// TIA Portal project "LABSDAMC" (V20)

(* hardware
DEVICE "S7-1500/ET200MP station_1"  S7-1500 station
   slot 0: "Rail_0"  Rack  6ES7 590-1***0-0AA0
   slot 1: "PLC_1"  CPU 1516-3 PN/DP  6ES7 516-3AN01-0AB0  V2.9
      slot 3: "CPU display_1"  6ES7591-1BA00-0AA0
      slot 32768: "PROFINET interface_1"  X1
         slot 32769: "Port_1"  X1 P1
         slot 32770: "Port_2"  X1 P2
      slot 33024: "PROFINET interface_2"  X2
         slot 33025: "Port_1"  X2 P1
      slot 33280: "DP interface_1"  X3
      slot 34817: "Virtual CP interface port_1"  Virtual CP interface port  Virtual CP interface port
   slot 2: "DI 32x24VDC HF_1"  DI 32x24VDC HF  6ES7 521-1BL00-0AB0  V2.2
   slot 3: "DQ 32x24VDC/0.5A HF_1"  DQ 32x24VDC/0.5A HF  6ES7 522-1BL01-0AB0  V1.1
   slot 4: "AI 8xU/I/RTD/TC ST_1"  AI 8xU/I/RTD/TC ST  6ES7 531-7KF00-0AB0  V2.2
   slot 5: "AQ 4xU/I ST_1"  AQ 4xU/I ST  6ES7 532-5HD00-0AB0  V2.2
DEVICE "HMI"  TP900 Comfort
   slot 0: "HMI"  TP900 Comfort  6AV2 124-0JC01-0AX0  17.0.0.0
   slot 1: "HMI_RT_1"  TP900 Comfort  6AV2 124-0JC01-0AX0  17.0.0.0
   slot 5: "HMI.IE_CP_1"  PROFINET Interface  17.0.0.0
      slot 1: "PROFINET Interface_1"  PROFINET Interface
         slot 1: "Port_1"  Port
         slot 2: "Port_2"  Port
   slot 7: "HMI.MPI/DP_CP_1"  MPI/DP Interface  17.0.0.0
*)

// ===== PLC "PLC_1"  CPU 1516-3 PN/DP =====

VAR_GLOBAL   // PLC tag table "Default tag table"
   "Conveyor_Start_Backward" AT %Q0.1 : Bool;
END_VAR

VAR_GLOBAL   // PLC tag table "Tags GRAPH Sequence"
   "GRAPH_Group_Fault" AT %M10.0 : Bool;
   "GRAPH_Count_Bottle" AT %MW12 : Int;
   "Valve_water" AT %Q1.1 : Bool;
   "Valve_AJC" AT %Q1.2 : Bool;
   "Valve_OJC" AT %Q1.3 : Bool;
   "GRAPH_Mixer_ON" AT %Q1.0 : Bool;
   "GRAPH_Start_Labeling" AT %Q2.0 : Bool;
   "GRAPH_Filling_Complete" AT %M20.0 : Bool;
   "Start_GRAPH_Sequence" AT %M100.0 : Bool;
END_VAR

VAR_GLOBAL   // PLC tag table "Tag-uri de umplere"
   "Valve_Fill_Bottle" AT %Q1.4 : Bool;
END_VAR

VAR_GLOBAL   // PLC tag table "Tag-uri transport"
   "Conveyor_Direction" AT %M0.1 : Bool;
   "Conveyor_Start_Conveyor" AT %M0.0 : Bool;
   "Conveyor_Drive_OK" AT %M0.2 : Bool;
   "Conveyor_Start_Forward" AT %Q0.0 : Bool;
END_VAR

VAR_GLOBAL   // PLC tag table "Tag-uri expirare"
   "Best_before_date" AT %MW2 : Int;
END_VAR

DATA_BLOCK "Global_DB"   // DB1
{ S7_Optimized_Access := 'TRUE' }
VERSION : 0.1
   VAR
      BBD_Duration : Int;
      Rețetă_element_concentrat_suc_de_mere : Time;
      Rețetă_element_concentrat_suc_orange : Time;
      Rețetă_element_apă : Time;
   END_VAR
BEGIN
END_DATA_BLOCK

DATA_BLOCK "SetareData"   // DB2
{ S7_Optimized_Access := 'TRUE' }
VERSION : 0.1
   VAR
      data : DTL;
      ok : Int;
      data_temp : DTL;
   END_VAR
BEGIN
END_DATA_BLOCK

DATA_BLOCK "SCL_Best_before_date_DB"   // DB4
{ S7_Optimized_Access := 'TRUE' }
VERSION : 0.1
// stored: InstanceOfName SCL_Best_before_date
"SCL_Best_before_date"
BEGIN
END_DATA_BLOCK

DATA_BLOCK "GRAPH_Sequence_DB_1"   // DB5
{ S7_Optimized_Access := 'TRUE' }
VERSION : 0.1
// stored: InstanceOfName GRAPH_Sequence
"GRAPH_Sequence"
BEGIN
END_DATA_BLOCK

FUNCTION_BLOCK "GRAPH_Sequence"   // FB1, GRAPH_PLUS
{ S7_Optimized_Access := 'TRUE' }
VERSION : 0.1
   VAR_INPUT
      OFF_SQ : Bool := false;   // Turn sequence off
      INIT_SQ : Bool := false;   // Set sequence to initial state
      ACK_EF : Bool := false;   // Acknowledge all errors and faults
      S_PREV : Bool := false;   // Output previous step in parameter S_NO
      S_NEXT : Bool := false;   // Indicate next step in parameter S_NO
      SW_AUTO : Bool := false;   // Automatic mode
      SW_TAP : Bool := false;   // Semiautomatic/switch with transition
      SW_TOP : Bool := false;   // Semiautomatic/ignore transition
      SW_MAN : Bool := false;   // Manual mode
      S_SEL : Int := 0;   // Select step to be output to S_NO
      S_ON : Bool := false;   // Activate step indicated in S_NO
      S_OFF : Bool := false;   // Disable step indicated in S_NO
      T_PUSH : Bool := false;   // Enable transition to switch in semi automatic mode
   END_VAR
   VAR_OUTPUT
      S_NO : Int := 0;   // Step number
      S_MORE : Bool := false;   // More steps are available and can be shown in S_NO
      S_ACTIVE : Bool := false;   // Step indicated in S_NO is active
      ERR_FLT : Bool := false;   // Interlock or supervision group error
      AUTO_ON : Bool := false;   // Automatic mode is active
      TAP_ON : Bool := false;   // Semiautomatic mode/step with transition enabled
      TOP_ON : Bool := false;   // Semiautomatic mode/ignore transition enabled
      MAN_ON : Bool := false;   // Manual mode is active
   END_VAR
   VAR
      HMI_INFO : Array[0..8] of UInt;
      IF_PAR : G7_IfParPlus_V6;
      RT_DATA : G7_RTDataPlus_V6;   // Internal data area
      Trans1 : G7_TransitionPlus_V6;   // Transition structure
      Trans2 : G7_TransitionPlus_V6;   // Transition structure
      Trans3 : G7_TransitionPlus_V6;   // Transition structure
      Trans4 : G7_TransitionPlus_V6;   // Transition structure
      Trans5 : G7_TransitionPlus_V6;   // Transition structure
      Trans6 : G7_TransitionPlus_V6;   // Transition structure
      Trans7 : G7_TransitionPlus_V6;   // Transition structure
      Trans8 : G7_TransitionPlus_V6;   // Transition structure
      Trans9 : G7_TransitionPlus_V6;   // Transition structure
      Home : G7_StepPlus_V6;   // Step structure
      "Umpleți ingredientele rețetei" : G7_StepPlus_V6;   // Step structure
      Mixer : G7_StepPlus_V6;   // Step structure
      "Transport de umplere" : G7_StepPlus_V6;   // Step structure
      Umplere : G7_StepPlus_V6;   // Step structure
      "Etichetarea transportului" : G7_StepPlus_V6;   // Step structure
      Etichetarea : G7_StepPlus_V6;   // Step structure
      "Umplere completă" : G7_StepPlus_V6;   // Step structure
      SINI : Array[0..1] of USInt;
      LSTT : Array[0..8] of USInt;
      ATAJ : Array[0..8] of USInt;
      ATAB : Array[0..8] of USInt;
      PSTT : Array[0..8] of USInt;
      NSTT : Array[0..8] of USInt;
      ASSJ : Array[0..7] of USInt;
      ASSB : Array[0..7] of USInt;
      PTTS : Array[0..7] of USInt;
      NTTS : Array[0..7] of USInt;
      SW_SQTS : Array[0..7] of USInt;
      SWITCH : Array[0..0] of USInt;
      TVX : Array[0..3] of USInt;
      TTX : Array[0..3] of USInt;
      TSX : Array[0..1] of USInt;
      S00X : Array[0..1] of USInt;
      SOFFX : Array[0..1] of USInt;
      SONX : Array[0..1] of USInt;
      SAX : Array[0..1] of USInt;
      SERRX : Array[0..8] of USInt;
      SMX : Array[0..8] of USInt;
      S0X : Array[0..8] of USInt;
      S1X : Array[0..8] of USInt;
      IL_ALARM_INST : Diag_Alarm;
      SUP_ALARM_INST : Diag_Alarm;
      STEP_TIME_ALARM_INST : Diag_Alarm;
      IEC_TIMER_INST : IEC_TIMER;
      TRANSACTION_FLAG : Bool := false;
   END_VAR
   // SINI[0] := 2;
   // LSTT[0] := 255;
   // LSTT[1] := 255;
   // LSTT[2] := 255;
   // LSTT[3] := 255;
   // LSTT[4] := 255;
   // LSTT[5] := 255;
   // LSTT[6] := 3;
   // LSTT[7] := 255;
   // ATAJ[1] := 1;
   // ATAJ[2] := 2;
   // ATAJ[3] := 3;
   // ATAJ[4] := 4;
   // ATAJ[5] := 5;
   // ATAJ[6] := 6;
   // ATAJ[7] := 7;
   // ATAJ[8] := 8;
   // ATAB[1] := 1;
   // ATAB[2] := 2;
   // ATAB[3] := 3;
   // ATAB[4] := 4;
   // ATAB[5] := 5;
   // ATAB[6] := 7;
   // ATAB[7] := 6;
   // ATAB[8] := 8;
   // PSTT[1] := 1;
   // PSTT[2] := 2;
   // PSTT[3] := 3;
   // PSTT[4] := 4;
   // PSTT[5] := 5;
   // PSTT[6] := 6;
   // PSTT[7] := 6;
   // PSTT[8] := 7;
   // NSTT[0] := 1;
   // NSTT[1] := 2;
   // NSTT[2] := 3;
   // NSTT[3] := 4;
   // NSTT[4] := 5;
   // NSTT[5] := 6;
   // NSTT[6] := 3;
   // NSTT[7] := 7;
   // ASSJ[1] := 1;
   // ASSJ[2] := 2;
   // ASSJ[3] := 3;
   // ASSJ[4] := 4;
   // ASSJ[5] := 5;
   // ASSJ[6] := 6;
   // ASSJ[7] := 7;
   // ASSB[1] := 1;
   // ASSB[2] := 2;
   // ASSB[3] := 3;
   // ASSB[4] := 4;
   // ASSB[5] := 5;
   // ASSB[6] := 6;
   // ASSB[7] := 7;
   // PTTS[0] := 255;
   // PTTS[2] := 1;
   // PTTS[3] := 2;
   // PTTS[4] := 3;
   // PTTS[5] := 4;
   // PTTS[6] := 5;
   // PTTS[7] := 7;
   // NTTS[1] := 1;
   // NTTS[2] := 2;
   // NTTS[3] := 3;
   // NTTS[4] := 4;
   // NTTS[5] := 5;
   // NTTS[6] := 6;
   // NTTS[7] := 8;
   // SW_SQTS[7] := 1;
   // TVX[0] := 16#1;
   // TTX[0] := 16#1;
   // TSX[0] := 16#1;
   // S00X[0] := 16#1;
   // SOFFX[0] := 16#1;
   // SONX[0] := 16#1;
   // SAX[0] := 16#1;
   // SERRX[0] := 16#1;
   // SMX[0] := 16#1;
   // S0X[0] := 16#1;
   // S1X[0] := 16#1;
BEGIN
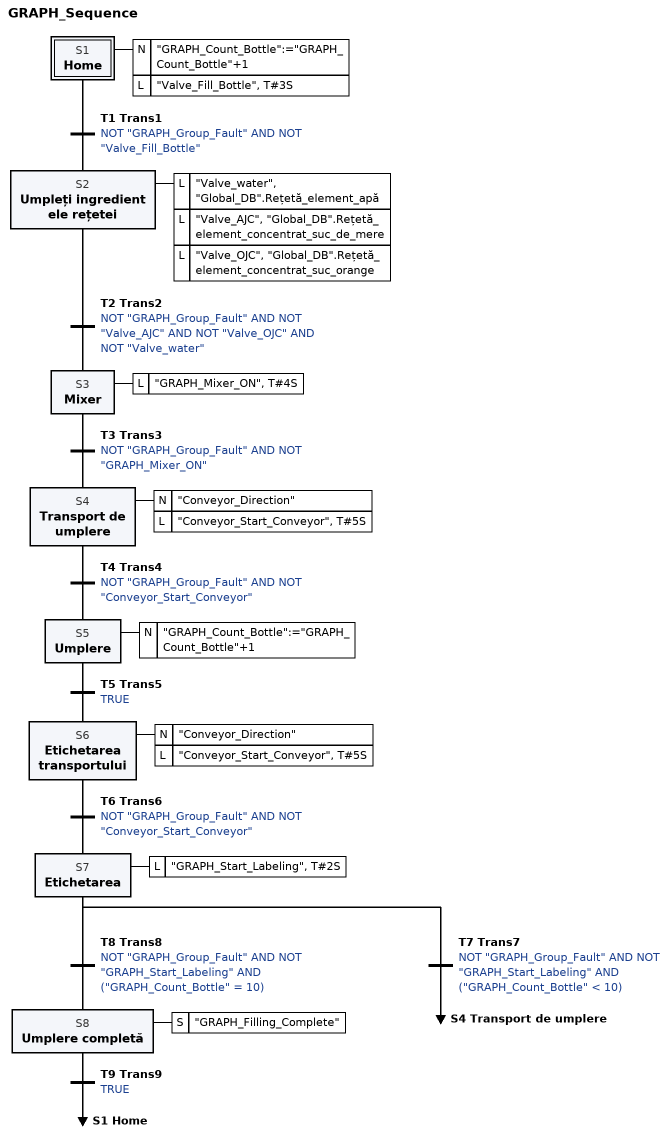
   // sequencer 1
   INITIAL_STEP Home:   // S1, max time T#10S, warning time T#7S
              N    "GRAPH_Count_Bottle":="GRAPH_Count_Bottle"+1
              L    "Valve_Fill_Bottle", T#3S
   END_STEP
   TRANSITION Trans1 FROM Home TO "Umpleți ingredientele rețetei"   // T1
      := NOT "GRAPH_Group_Fault" AND NOT "Valve_Fill_Bottle";
   END_TRANSITION
   STEP "Umpleți ingredientele rețetei":   // S2, max time T#10S, warning time T#7S
              L    "Valve_water", "Global_DB".Rețetă_element_apă
              L    "Valve_AJC", "Global_DB".Rețetă_element_concentrat_suc_de_mere
              L    "Valve_OJC", "Global_DB".Rețetă_element_concentrat_suc_orange
   END_STEP
   TRANSITION Trans2 FROM "Umpleți ingredientele rețetei" TO Mixer   // T2
      := NOT "GRAPH_Group_Fault" AND NOT "Valve_AJC" AND NOT "Valve_OJC" AND NOT "Valve_water";
   END_TRANSITION
   STEP Mixer:   // S3, max time T#10S, warning time T#7S
              L    "GRAPH_Mixer_ON", T#4S
   END_STEP
   TRANSITION Trans3 FROM Mixer TO "Transport de umplere"   // T3
      := NOT "GRAPH_Group_Fault" AND NOT "GRAPH_Mixer_ON";
   END_TRANSITION
   STEP "Transport de umplere":   // S4, max time T#10S, warning time T#7S
              N    "Conveyor_Direction"
              L    "Conveyor_Start_Conveyor", T#5S
   END_STEP
   TRANSITION Trans4 FROM "Transport de umplere" TO Umplere   // T4
      := NOT "GRAPH_Group_Fault" AND NOT "Conveyor_Start_Conveyor";
   END_TRANSITION
   STEP Umplere:   // S5, max time T#10S, warning time T#7S
              N    "GRAPH_Count_Bottle":="GRAPH_Count_Bottle"+1
   END_STEP
   TRANSITION Trans5 FROM Umplere TO "Etichetarea transportului"   // T5
      := TRUE;
   END_TRANSITION
   STEP "Etichetarea transportului":   // S6, max time T#10S, warning time T#7S
              N    "Conveyor_Direction"
              L    "Conveyor_Start_Conveyor", T#5S
   END_STEP
   TRANSITION Trans6 FROM "Etichetarea transportului" TO Etichetarea   // T6
      := NOT "GRAPH_Group_Fault" AND NOT "Conveyor_Start_Conveyor";
   END_TRANSITION
   STEP Etichetarea:   // S7, max time T#10S, warning time T#7S
              L    "GRAPH_Start_Labeling", T#2S
   END_STEP
   TRANSITION Trans8 FROM Etichetarea TO "Umplere completă"   // T8
      := NOT "GRAPH_Group_Fault" AND NOT "GRAPH_Start_Labeling" AND ("GRAPH_Count_Bottle" = 10);
   END_TRANSITION
   TRANSITION Trans7 FROM Etichetarea TO "Transport de umplere"   // T7, jump
      := NOT "GRAPH_Group_Fault" AND NOT "GRAPH_Start_Labeling" AND ("GRAPH_Count_Bottle" < 10);
   END_TRANSITION
   STEP "Umplere completă":   // S8, max time T#10S, warning time T#7S
              S    "GRAPH_Filling_Complete"
   END_STEP
   TRANSITION Trans9 FROM "Umplere completă" TO Home   // T9, jump
      := TRUE;
   END_TRANSITION
END_FUNCTION_BLOCK

FUNCTION_BLOCK "SCL_Best_before_date"   // FB2, SCL
{ S7_Optimized_Access := 'TRUE' }
VERSION : 0.1
   VAR_INPUT
      Duration : Int;
   END_VAR
   VAR_OUTPUT
      Best_before_date_Output : Int;
   END_VAR
   VAR_TEMP
      Error : Int;
      System_Time_DT : DTL;
   END_VAR
BEGIN
   #Error := RD_SYS_T(OUT => #System_Time_DT);
   #Best_before_date_Output := "SetareData".data_temp.YEAR + #Duration;
END_FUNCTION_BLOCK

FUNCTION "STL-Conveyor" : Void   // FC1, STL
{ S7_Optimized_Access := 'TRUE' }
VERSION : 0.1
   VAR_INPUT
      START_INPUT : Bool;
      Direction : Bool;
   END_VAR
   VAR_OUTPUT
      Conveyor_DONE : Bool;
      Forward : Bool;
      Backward : Bool;
   END_VAR
BEGIN

REGION Network 1
         A     #Direction;
         A     #START_INPUT;
         S     #Forward;
         R     #Conveyor_DONE;
END_REGION

REGION Network 2
         AN    #Direction;
         A     #START_INPUT;
         S     #Backward;
         R     #Conveyor_DONE;
END_REGION

REGION Network 3
         AN    #Direction;
         R     #Forward;
         R     #Backward;
         S     #Conveyor_DONE;
END_REGION
END_FUNCTION

ORGANIZATION_BLOCK "Main"   // OB1, LAD, ProgramCycle
TITLE = "Main Program Sweep (Cycle)"
{ S7_Optimized_Access := 'TRUE' }
VERSION : 0.1
   VAR_INPUT
      Initial_Call : Bool;   // Initial call of this OB
      Remanence : Bool;   // =True, if remanent data are available
   END_VAR
BEGIN

REGION Network 1
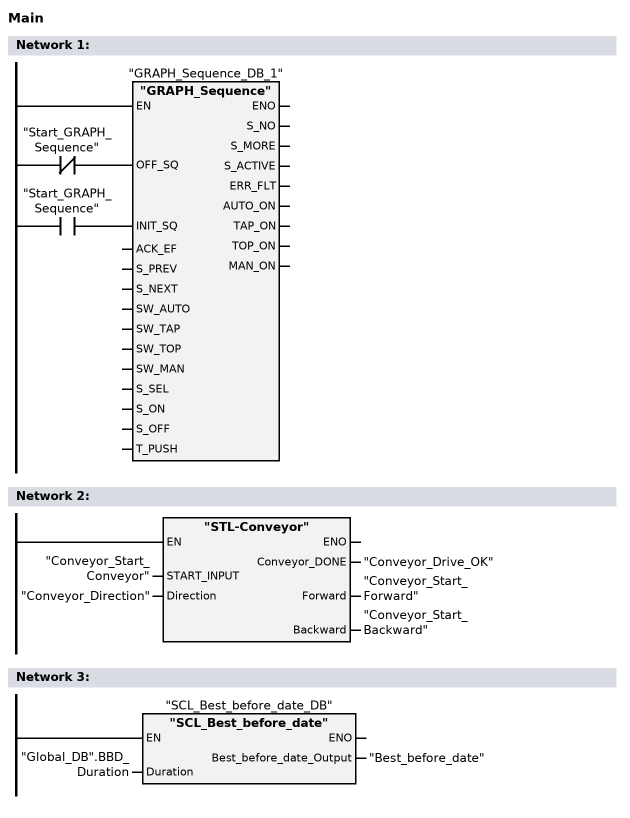
   RUNG wire#powerrail
      "GRAPH_Sequence_DB_1"(OFF_SQ := wire#w1, INIT_SQ := wire#w2, ACK_EF :=, S_PREV :=, S_NEXT :=, SW_AUTO :=, SW_TAP :=, SW_TOP :=, SW_MAN :=, S_SEL :=, S_ON :=, S_OFF :=, T_PUSH :=, S_NO =>, S_MORE =>, S_ACTIVE =>, ERR_FLT =>, AUTO_ON =>, TAP_ON =>, TOP_ON =>, MAN_ON =>)
   END_RUNG
   RUNG wire#powerrail
      I_Contact( "Start_GRAPH_Sequence" )
   END_RUNG wire#w1
   RUNG wire#powerrail
      Contact( "Start_GRAPH_Sequence" )
   END_RUNG wire#w2
   // the same network as SCL:
   "GRAPH_Sequence_DB_1"(OFF_SQ := NOT "Start_GRAPH_Sequence", INIT_SQ := "Start_GRAPH_Sequence");   // "GRAPH_Sequence"
END_REGION

REGION Network 2
   RUNG wire#powerrail
      "STL-Conveyor"(START_INPUT := "Conveyor_Start_Conveyor", Direction := "Conveyor_Direction", Conveyor_DONE => "Conveyor_Drive_OK", Forward => "Conveyor_Start_Forward", Backward => "Conveyor_Start_Backward")
   END_RUNG
   // the same network as SCL:
   "STL-Conveyor"(START_INPUT := "Conveyor_Start_Conveyor",
                  Direction := "Conveyor_Direction",
                  Conveyor_DONE => "Conveyor_Drive_OK",
                  Forward => "Conveyor_Start_Forward",
                  Backward => "Conveyor_Start_Backward");
END_REGION

REGION Network 3
   RUNG wire#powerrail
      "SCL_Best_before_date_DB"(Duration := "Global_DB".BBD_Duration, Best_before_date_Output => "Best_before_date")
   END_RUNG
   // the same network as SCL:
   "SCL_Best_before_date_DB"(Duration := "Global_DB".BBD_Duration,   // "SCL_Best_before_date"
                           Best_before_date_Output => "Best_before_date");
END_REGION
END_ORGANIZATION_BLOCK

(* ===== HMI "HMI_RT_1" =====
system functions are stored by id; their names below are inferred from use
connection "HMI_Connection_1": ETHERNET, S7_1500_OMS

HMI tags "Default tag table"
   "Tag_ScreenNumber" : UInt, internal
   "GRAPH_Sequence_DB_1_Mixer_X" : Bool = PLC GRAPH_Sequence_DB_1.Mixer.X, 1 s
   "Position_Bottle" : Int, internal
   "GRAPH_Sequence_DB_1_Transport de umplere_X" : Bool = PLC GRAPH_Sequence_DB_1."Transport de umplere".X, 1 s
      on ChangeValue: SetTag("Position_Bottle", 0)
   "GRAPH_Sequence_DB_1_Umplere_X" : Bool = PLC GRAPH_Sequence_DB_1.Umplere.X, 1 s
   "Position_Bottle_1" : Int, internal
   "GRAPH_Sequence_DB_1_Etichetarea transportului_X" : Bool = PLC GRAPH_Sequence_DB_1."Etichetarea transportului".X, 1 s
      on ChangeValue: SetTag("Position_Bottle_1", 0)
   "GRAPH Sequence_DB_Transport Filling.X" : Bool = PLC GRAPH_Sequence_DB_1."Transport de umplere".X AT %DB1.DBX0.0, 1 s
      on ChangeValue: SetTag("Position_Bottle", 0)
   "GRAPH_Count_Bottle" : Int = PLC GRAPH_Count_Bottle AT %MW12, 1 s
   "GRAPH_Sequence_DB_1_Umpleți ingredientele rețetei_X" : Bool = PLC GRAPH_Sequence_DB_1."Umpleți ingredientele rețetei".X, 1 s
   "GRAPH_Sequence_DB_1_Etichetarea_X" : Bool = PLC GRAPH_Sequence_DB_1.Etichetarea.X, 1 s
   "Best_before_date" : Int = PLC Best_before_date AT %MW2, 1 s
   "Start_GRAPH_Sequence" : Bool = PLC Start_GRAPH_Sequence AT %M100.0, 1 s
   "Global_DB_Rețetă_element_apă" : Time = PLC Global_DB.Rețetă_element_apă, 1 s
   "Global_DB_Rețetă_element_concentrat_suc_de_mere" : Time = PLC Global_DB.Rețetă_element_concentrat_suc_de_mere, 1 s
   "Global_DB_Rețetă_element_concentrat_suc_orange" : Time = PLC Global_DB.Rețetă_element_concentrat_suc_orange, 1 s

recipe "Recipe_Beverage": Water <- "Global_DB_Rețetă_element_apă", "Concentrate_Apple_Juice <- "Global_DB_Rețetă_element_concentrat_suc_de_mere", "Concentrate_Orange_Juice <- "Global_DB_Rețetă_element_concentrat_suc_orange"

screen "Production" 800x420, template "Template_1"
   on GenerateScreen: SetTag("Tag_ScreenNumber", 1); function_f9c01323("Position_Bottle", 1, 50, 0, 2); function_f9c01323("Position_Bottle_1", 1, 50, 0, 2)
   Button "HmiScreenItemData" at 217,9 size 159x47; TextOff 'Recipes'; PictureOff "Navigates to Recipes for TP900 Comfort 17.0.0.0"; PictureOn "Navigates to Recipes for TP900 Comfort 17.0.0.0"
      on Release: ActivateScreen("Recipes", 0)
   Button "HmiScreenItemData_1" at 407,9 size 159x47; TextOff 'Diagnostics view'; PictureOff "Navigates to Diagnostics view for TP900 Comfort 17.0.0.0"; PictureOn "Navigates to Diagnostics view for TP900 Comfort 17.0.0.0"
      on Release: ActivateScreen("Diagnostics view", 0)
   Button "HmiScreenItemData_3" at 36,10 size 159x47; TextOff 'System screens'; PictureOff "Navigates to System screens for TP900 Comfort 17.0.0.0"; PictureOn "Navigates to System screens for TP900 Comfort 17.0.0.0"
      on Release: ActivateScreen("System screens", 0)
   GraphicView "Graphic view_1" at 157,267 size 590x82; Picture "Graphic_2"
   GraphicView "Graphic view_2" at 432,134 size 64x121; Picture "Graphic_3"
   GraphicView "Graphic view_5" at 180,87 size 27x42; Picture "Graphic_5"
   GraphicView "Graphic view_4" at 230,87 size 27x42; Picture "Graphic_5"
   GraphicView "Graphic view_6" at 282,87 size 27x42; Picture "Graphic_5"
   GraphicView "Graphic view_8" at 189,122 size 10x47; Picture "Graphic_7"
   GraphicView "Graphic view_7" at 238,122 size 10x47; Picture "Graphic_7"
   GraphicView "Graphic view_9" at 291,122 size 10x47; Picture "Graphic_7"
   GraphicView "Graphic view_10" at 180,160 size 271x15; Picture "Graphic_8"
   GraphicView "Graphic view_3" at 449,145 size 33x34; Picture "Graphic_4"
      Appearance <- "GRAPH_Sequence_DB_1_Mixer_X"
   GraphicView "Graphic view_11" at 263,256 size 19x50; Picture "Graphic_11"
      HorizontalMovement <- "Position_Bottle"
      Visibility <- "GRAPH_Sequence_DB_1_Transport de umplere_X"
   GraphicView "Graphic view_12" at 455,257 size 19x50; Picture "Graphic_11"
      Visibility <- "GRAPH_Sequence_DB_1_Umplere_X"
   GraphicView "Graphic view_13" at 455,258 size 19x50; Picture "Graphic_11"
      HorizontalMovement <- "Position_Bottle_1"
      Visibility <- "GRAPH_Sequence_DB_1_Etichetarea transportului_X"
   Bar "Bar_1" at 508,146 size 68x98; MinimumValue 0; MaximumValue 10
      ProcessValue <- "GRAPH_Count_Bottle"
   Circle "Circle_1" at 327,113 size 26x26
      Appearance <- "GRAPH_Sequence_DB_1_Umpleți ingredientele rețetei_X"
   Circle "Circle_2" at 579,183 size 26x26
      Appearance <- "GRAPH Sequence_DB_Transport Filling.X"
   Rectangle "Rectangle_1" at 638,223 size 15x49
      Appearance <- "GRAPH_Sequence_DB_1_Etichetarea_X"
   IOField "I/O field_1" at 668,243 size 96x32; FormatPattern 9999
      ProcessValue <- "Best_before_date"
   Switch "Rotary_RG" at 650,98 size 80x80; CaptionText 'Switch'; TextOff '0'; TextOn '1'; PictureOn "Rotary_RG_On_256c"; PictureOff "Rotary_RG_Off_256c"
      ProcessValue <- "Start_GRAPH_Sequence"
   TextField "Text field_1" at 216,64 size 91x20; Text 'Ingredients'
   TextField "Text field_3" at 438,110 size 153x20; Text 'Filling station/Mixer'
   TextField "Text field_4" at 644,193 size 124x20; Text 'Labeling station'
   TextField "Text field_5" at 668,212 size 92x20; Text 'Best before'

Template "Template_1" 800x420
   Button "Template_Button" at 720,360 size 78x58; TextOff 'Text'
   Button "Template_Button_1" at 640,360 size 78x58; TextOff 'Text'
   Button "Template_Button_2" at 560,360 size 78x58; TextOff 'Text'
   Button "Template_Button_3" at 480,360 size 78x58; TextOff 'Text'
   Button "Template_Button_4" at 400,360 size 78x58; TextOff 'Text'
   Button "Template_Button_5" at 321,360 size 78x58; TextOff 'Text'
   Button "Template_Button_6" at 241,360 size 78x58; TextOff 'Text'
   Button "Template_Button_7" at 161,360 size 78x58; TextOff 'Text'
   Button "Alarms" at 81,360 size 78x58; TextOff 'Alarms'; PictureOff "AlarmDisplay_TP900_Comfort_TR"; PictureOn "AlarmDisplay_TP900_Comfort_TR"
      on Release: function_ef3f5d25("Alarm window_Unacknowledged", -1)
   Button "Template_Button_8" at 1,360 size 78x58; TextOff 'Text'
   GraphicView "Template_Graphic view_1" at 7,365 size 61x53; Picture "Graphic_9"
   GraphicView "Template_Graphic view_2" at 734,365 size 50x52; Picture "Graphic_10"

screen "Recipes" 800x420, template "Template_1"
   on GenerateScreen: SetTag("Tag_ScreenNumber", 2)
   TextField "HmiScreenItemData" at 80,167 size 640x22; Text 'Recipes'
   Button "Back" at 1,1 size 159x47; TextOff 'Back'
      on Release: ActivateScreen("Production", 0)

screen "Diagnostics view" 800x420, template "Template_1"
   on GenerateScreen: SetTag("Tag_ScreenNumber", 3)
   TextField "HmiScreenItemData" at 80,167 size 640x22; Text 'Diagnostics view'
   Button "Back" at 1,1 size 159x47; TextOff 'Back'
      on Release: ActivateScreen("Production", 0)

screen "System screens" 800x420, template "Template_1"
   on GenerateScreen: SetTag("Tag_ScreenNumber", 4)
   Button "Back" at 1,1 size 159x47; TextOff 'Back'
      on Release: ActivateScreen("Production", 0)
   Button "HmiScreenItemData" at 36,95 size 159x47; TextOff 'SIMATIC PLC watch table'; PictureOff "Navigates to SIMATIC PLC watch table for TP900 Comfort 17.0.0.0"; PictureOn "Navigates to SIMATIC PLC watch table for TP900 Comfort 17.0.0.0"
      on Release: ActivateScreen("SIMATIC PLC watch table", 0)
   Button "HmiScreenItemData_1" at 36,154 size 159x47; TextOff 'Project information'; PictureOff "Navigates to Project information for TP900 Comfort 17.0.0.0"; PictureOn "Navigates to Project information for TP900 Comfort 17.0.0.0"
      on Release: ActivateScreen("Project information", 0)
   Button "HmiScreenItemData_2" at 36,213 size 159x47; TextOff 'System settings'; PictureOff "Navigates to System settings for TP900 Comfort 17.0.0.0"; PictureOn "Navigates to System settings for TP900 Comfort 17.0.0.0"
      on Release: ActivateScreen("System settings", 0)
   Button "HmiScreenItemData_3" at 36,272 size 159x47; TextOff 'User administration'; PictureOff "Navigates to User administration for TP900 Comfort 17.0.0.0"; PictureOn "Navigates to User administration for TP900 Comfort 17.0.0.0"
      on Release: ActivateScreen("User administration", 0)
   Button "HmiScreenItemData_4" at 207,95 size 159x47; TextOff 'System information'; PictureOff "Navigates to System information for TP900 Comfort 17.0.0.0"; PictureOn "Navigates to System information for TP900 Comfort 17.0.0.0"
      on Release: ActivateScreen("System information", 0)
   Button "HmiScreenItemData_5" at 207,154 size 159x47; TextOff 'Different jobs'; PictureOff "Navigates to Different jobs for TP900 Comfort 17.0.0.0"; PictureOn "Navigates to Different jobs for TP900 Comfort 17.0.0.0"
      on Release: ActivateScreen("Different jobs", 0)

screen "SIMATIC PLC watch table" 800x420, template "Template_1"
   on GenerateScreen: SetTag("Tag_ScreenNumber", 5)
   StatusForce "HmiScreenItemData" at 1,49 size 796x304; ToolTipText 'Text'
   Button "Back" at 1,1 size 159x47; TextOff 'Back'
      on Release: ActivateScreen("System screens", 0)

screen "Project information" 800x420, template "Template_1"
   on GenerateScreen: SetTag("Tag_ScreenNumber", 6)
   TextField "HmiScreenItemData" at 35,51 size 171x28; Text 'Project name:'
   TextField "HmiScreenItemData_1" at 241,51 size 524x28; Text 'LABSDAMC'
   TextField "HmiScreenItemData_2" at 35,81 size 171x28; Text 'Created on:'
   TextField "HmiScreenItemData_3" at 241,81 size 524x28; Text '10/30/2025 12:12:25 PM'
   TextField "HmiScreenItemData_4" at 35,111 size 171x28; Text 'Author:'
   TextField "HmiScreenItemData_5" at 241,111 size 524x28; Text 'P4P4D13'
   TextField "HmiScreenItemData_6" at 35,141 size 171x28; Text 'Description:'
   TextField "HmiScreenItemData_7" at 241,141 size 524x28; Text '(not configured)'
   Button "Back" at 1,1 size 159x47; TextOff 'Back'
      on Release: ActivateScreen("System screens", 0)

screen "System settings" 800x420, template "Template_1"
   on GenerateScreen: SetTag("Tag_ScreenNumber", 7)
   Button "Calibrate screen" at 36,95 size 159x47; TextOff 'Calibrate screen'
      on Release: function_bc3e350c()
   Button "Clean screen" at 36,154 size 159x47; TextOff 'Clean screen'
      on Release: function_be740847(30)
   Button "Back" at 1,1 size 159x47; TextOff 'Back'
      on Release: ActivateScreen("System screens", 0)

screen "User administration" 800x420, template "Template_1"
   on GenerateScreen: SetTag("Tag_ScreenNumber", 8)
   UserView "HmiScreenItemData" at 1,49 size 796x304
   Button "Back" at 1,1 size 159x47; TextOff 'Back'
      on Release: ActivateScreen("System screens", 0)

screen "System information" 800x420, template "Template_1"
   on GenerateScreen: SetTag("Tag_ScreenNumber", 9)
   TextField "HmiScreenItemData" at 35,51 size 171x28; Text 'HMI device type:'
   TextField "HmiScreenItemData_1" at 241,51 size 524x28; Text 'TP900 Comfort 17.0.0.0'
   TextField "HmiScreenItemData_2" at 35,81 size 171x28; Text 'Version:'
   TextField "HmiScreenItemData_3" at 35,111 size 171x28; Text 'Connection:'
   TextField "HmiScreenItemData_4" at 241,111 size 524x28; Text '(not configured)'
   TextField "HmiScreenItemData_5" at 35,141 size 171x28; Text 'PLC:'
   TextField "HmiScreenItemData_6" at 241,141 size 524x28; Text '<PLC>'
   Button "Display version" at 241,81 size 524x28; TextOff 'Display version'
      on Release: function_febcb963(-1)
   Button "Back" at 1,1 size 159x47; TextOff 'Back'
      on Release: ActivateScreen("System screens", 0)

screen "Different jobs" 800x420, template "Template_1"
   on GenerateScreen: SetTag("Tag_ScreenNumber", 10)
   Button "Online" at 36,95 size 159x47; TextOff 'Online'
      on Release: function_bb44b551(0)
   Button "Offline" at 36,154 size 159x47; TextOff 'Offline'
      on Release: function_bb44b551(1)
   Button "Transfer" at 36,213 size 159x47; TextOff 'Transfer'
      on Release: function_bb44b551(2)
   Button "Toggle language" at 36,272 size 159x47; TextOff 'Toggle language'
      on Release: function_fb9197e8(-1)
   Button "Control Panel" at 207,95 size 159x47; TextOff 'Control Panel'
      on Release: function_f34a74f3()
   Button "Stop Runtime" at 207,154 size 159x47; TextOff 'Stop Runtime'
      on Release: StopRuntime(0)
   Button "Back" at 1,1 size 159x47; TextOff 'Back'
      on Release: ActivateScreen("System screens", 0)
*)